TYPE stLaserMachine EXTENDS stPimMachineData :
STRUCT
	
END_STRUCT
END_TYPE

(* stored: Version 1.1.0.1, ProductVersion 3.1.4024.13
   DUT stLaserMachine: Id {5e345f25-5cda-4823-914d-fd588fcf5081} *)
